// TIA Portal V20 export
TYPE "LBP_typePowerrideConfig"
TITLE = Data type for configuration of Powerride / Type de données pour la configuration Powerride
// User data type for LBP_PowerrideConfig / Type de données utilisateur pour LBP_PowerrideConfig
   STRUCT
      pos100 { S7_SetPoint := 'True'} : USInt := 0;   // [1..36] switch position at 100% ovr / [1..36] position du commutateur à correction 100 %
      posMax { S7_SetPoint := 'True'} : USInt := 0;   // [1..36] switch position at maximum ovr / [1..36] position du commutateur à correction maximale
      delay100 { S7_SetPoint := 'True'} : Time := T#500MS;   // time delay at 100% before continuing ovr / délai à 100 % avant de continuer correction
      switchPos { S7_SetPoint := 'True'} : Array[1..36] of "LBP_typePowerrideConfigPos";   // value, colour and vibration for position / valeur, couleur et vibration pour la position
   END_STRUCT;
END_TYPE
